{attribute 'qualified_only'}
TYPE EProductTypes :
(
	none := 0,
	unknown := 1,
	
	white := 2,
	black := 3,
	metal := 4
) UINT;
END_TYPE

(* stored: Version 1.1.0.1
   DUT EProductTypes: Id {df48ec1b-937a-4320-b603-b4a9227f010a} *)
